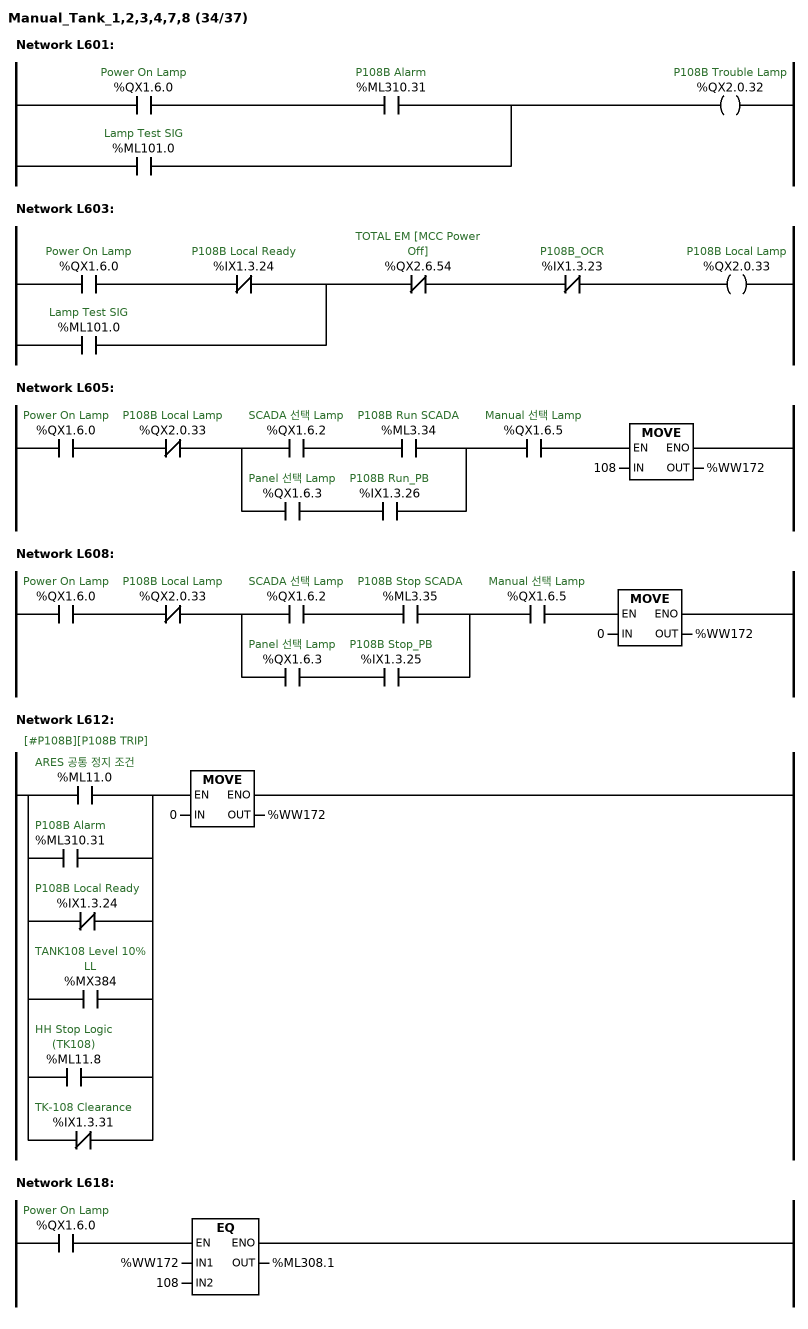
(* [picture p48: Manual_Tank_1,2,3,4,7,8 rungs L601-L618] *)
(* Rung L601 *)
%QX2.0.32 := (%QX1.6.0 AND %ML310.31) OR %ML101.0;
(* Rung L603 *)
%QX2.0.33 := ((%QX1.6.0 AND NOT %IX1.3.24) OR %ML101.0) AND NOT %QX2.6.54 AND NOT %IX1.3.23;
(* Rung L605 *)
IF %QX1.6.0 AND NOT %QX2.0.33 AND ((%QX1.6.2 AND %ML3.34) OR (%QX1.6.3 AND %IX1.3.26)) AND %QX1.6.5 THEN
    %WW172 := 108;
END_IF;
(* Rung L608 *)
IF %QX1.6.0 AND NOT %QX2.0.33 AND ((%QX1.6.2 AND %ML3.35) OR (%QX1.6.3 AND %IX1.3.25)) AND %QX1.6.5 THEN
    %WW172 := 0;
END_IF;
(* [#P108B][P108B TRIP] *)
(* Rung L612 *)
IF %ML11.0 OR %ML310.31 OR NOT %IX1.3.24 OR %MX384 OR %ML11.8 OR NOT %IX1.3.31 THEN %WW172 := 0; END_IF;
(* Rung L618 *)
IF %QX1.6.0 THEN %ML308.1 := %WW172 = 108; END_IF;

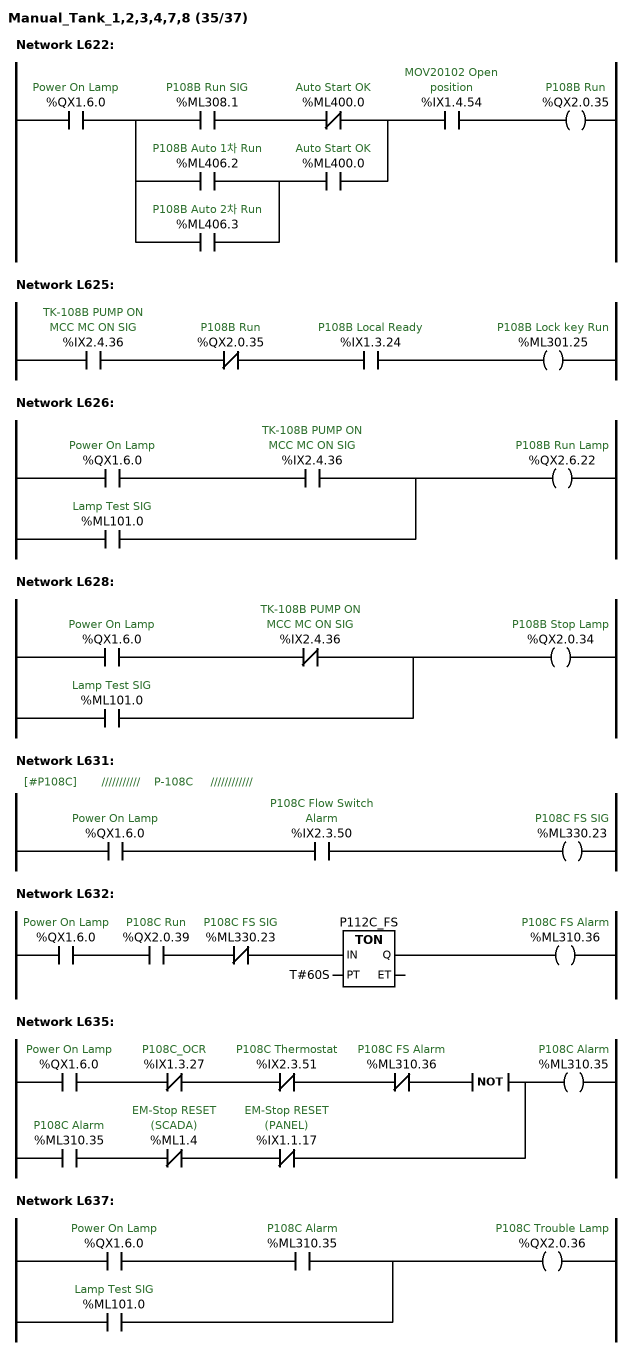
(* Rung L622 *)
%QX2.0.35 := %QX1.6.0 AND ((%ML308.1 AND NOT %ML400.0) OR ((%ML406.2 OR %ML406.3) AND %ML400.0)) AND %IX1.4.54;
(* Rung L625 *)
%ML301.25 := %IX2.4.36 AND NOT %QX2.0.35 AND %IX1.3.24;
(* Rung L626 *)
%QX2.6.22 := (%QX1.6.0 AND %IX2.4.36) OR %ML101.0;
(* Rung L628 *)
%QX2.0.34 := (%QX1.6.0 AND NOT %IX2.4.36) OR %ML101.0;
(* [#P108C]       ///////////    P-108C     //////////// *)
(* Rung L631 *)
%ML330.23 := %QX1.6.0 AND %IX2.3.50;
(* Rung L632 *)
P112C_FS(IN := %QX1.6.0 AND %QX2.0.39 AND NOT %ML330.23, PT := T#60S);
%ML310.36 := P112C_FS.Q;
(* Rung L635 *)
%ML310.35 := NOT (%QX1.6.0 AND NOT %IX1.3.27 AND NOT %IX2.3.51 AND NOT %ML310.36) OR (%ML310.35 AND NOT %ML1.4 AND NOT %IX1.1.17);
(* Rung L637 *)
%QX2.0.36 := (%QX1.6.0 AND %ML310.35) OR %ML101.0;

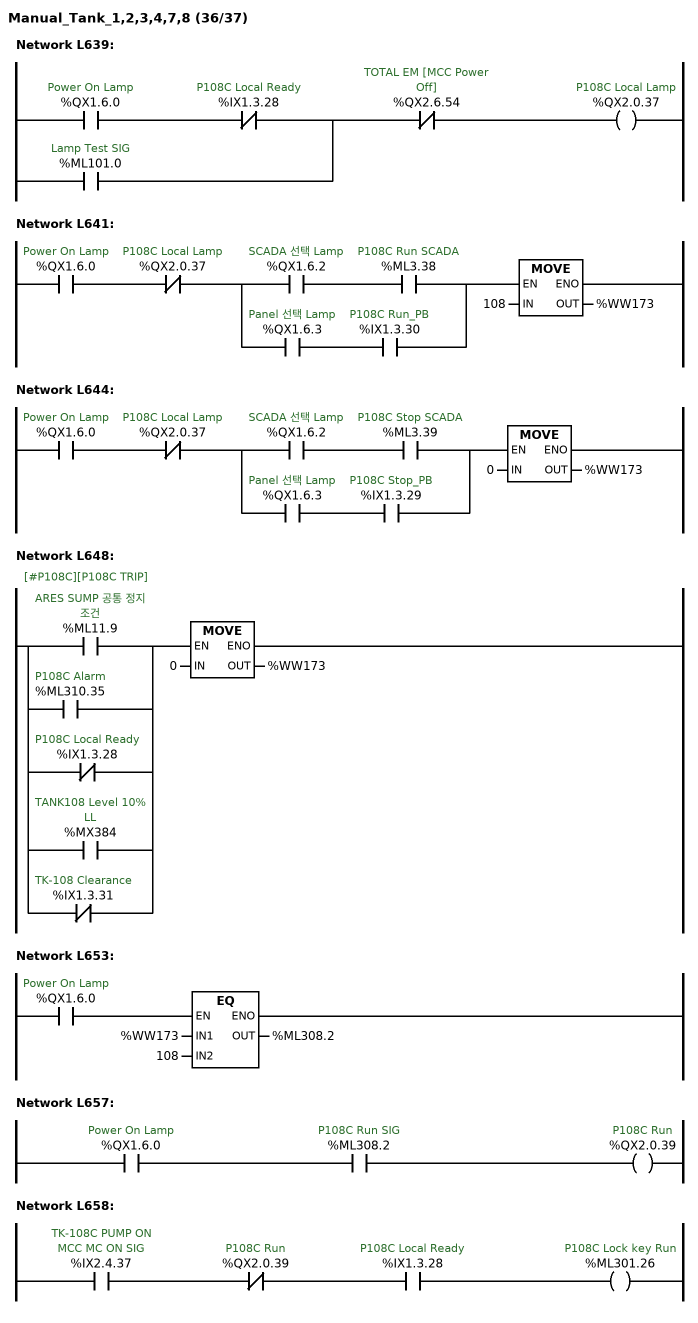
(* Rung L639 *)
%QX2.0.37 := ((%QX1.6.0 AND NOT %IX1.3.28) OR %ML101.0) AND NOT %QX2.6.54;
(* Rung L641 *)
IF %QX1.6.0 AND NOT %QX2.0.37 AND ((%QX1.6.2 AND %ML3.38) OR (%QX1.6.3 AND %IX1.3.30)) THEN
    %WW173 := 108;
END_IF;
(* Rung L644 *)
IF %QX1.6.0 AND NOT %QX2.0.37 AND ((%QX1.6.2 AND %ML3.39) OR (%QX1.6.3 AND %IX1.3.29)) THEN
    %WW173 := 0;
END_IF;
(* [#P108C][P108C TRIP] *)
(* Rung L648 *)
IF %ML11.9 OR %ML310.35 OR NOT %IX1.3.28 OR %MX384 OR NOT %IX1.3.31 THEN %WW173 := 0; END_IF;
(* Rung L653 *)
IF %QX1.6.0 THEN %ML308.2 := %WW173 = 108; END_IF;
(* Rung L657 *)
%QX2.0.39 := %QX1.6.0 AND %ML308.2;
(* Rung L658 *)
%ML301.26 := %IX2.4.37 AND NOT %QX2.0.39 AND %IX1.3.28;

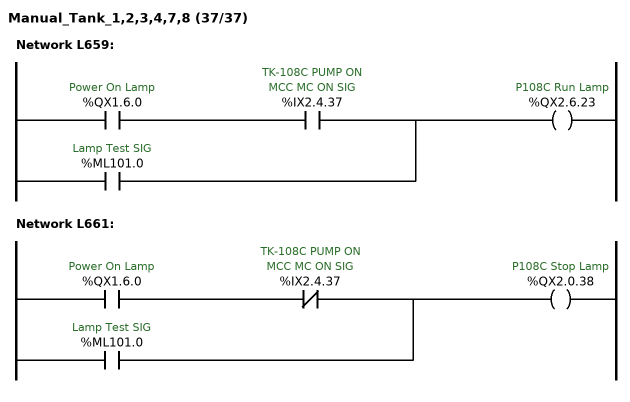
(* Rung L659 *)
%QX2.6.23 := (%QX1.6.0 AND %IX2.4.37) OR %ML101.0;
(* Rung L661 *)
%QX2.0.38 := (%QX1.6.0 AND NOT %IX2.4.37) OR %ML101.0;
END_PROGRAM

PROGRAM Manual_Tank_5,6,9,10 (* task: 스캔 프로그램 *)
VAR
    P105A_FS : TON;
    P105B_FS : TON;
    P105C_FS : TON;
    P106A_FS : TON;
    P106B_FS : TON;
    P106C_FS : TON;
    P109A_FS : TON;
    P109B_FS : TON;
    P109C_FS : TON;
    P110A_FS : TON;
    P110B_FS : TON;
    P110C_FS : TON;
END_VAR

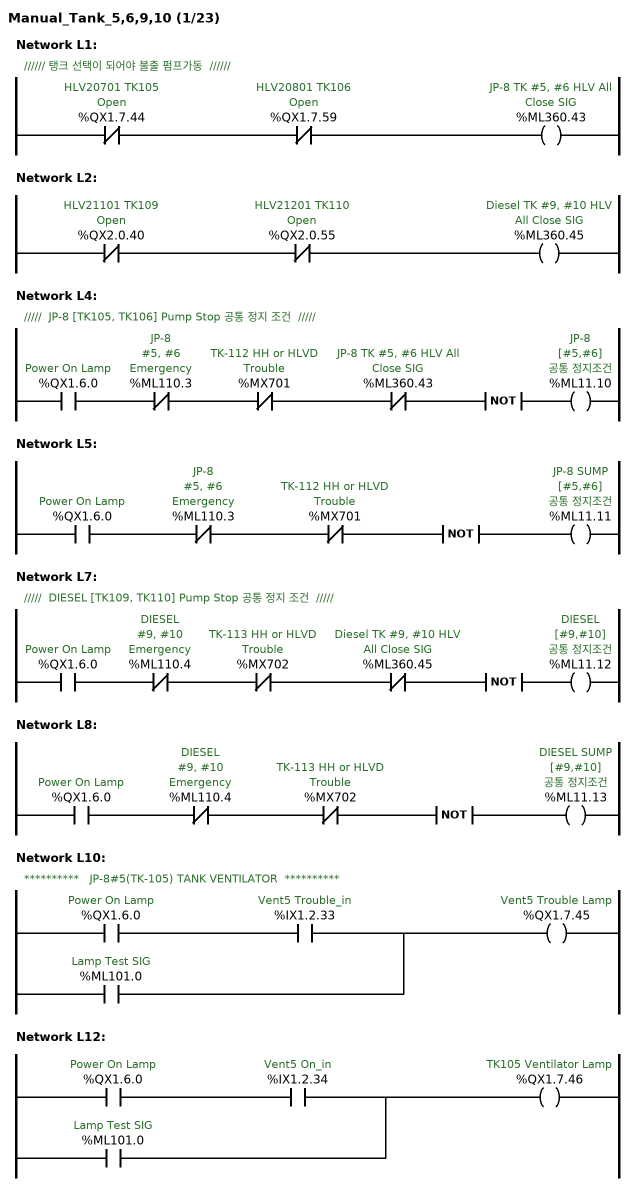
(* ////// 탱크 선택이 되어야 불출 펌프가동  ////// *)
(* Rung L1 *)
%ML360.43 := NOT %QX1.7.44 AND NOT %QX1.7.59;
(* Rung L2 *)
%ML360.45 := NOT %QX2.0.40 AND NOT %QX2.0.55;
(* /////  JP-8 [TK105, TK106] Pump Stop 공통 정지 조건  ///// *)
(* Rung L4 *)
%ML11.10 := NOT (%QX1.6.0 AND NOT %ML110.3 AND NOT %MX701 AND NOT %ML360.43);
(* Rung L5 *)
%ML11.11 := NOT (%QX1.6.0 AND NOT %ML110.3 AND NOT %MX701);
(* /////  DIESEL [TK109, TK110] Pump Stop 공통 정지 조건  ///// *)
(* Rung L7 *)
%ML11.12 := NOT (%QX1.6.0 AND NOT %ML110.4 AND NOT %MX702 AND NOT %ML360.45);
(* Rung L8 *)
%ML11.13 := NOT (%QX1.6.0 AND NOT %ML110.4 AND NOT %MX702);
(* **********   JP-8#5(TK-105) TANK VENTILATOR  ********** *)
(* Rung L10 *)
%QX1.7.45 := (%QX1.6.0 AND %IX1.2.33) OR %ML101.0;
(* Rung L12 *)
%QX1.7.46 := (%QX1.6.0 AND %IX1.2.34) OR %ML101.0;

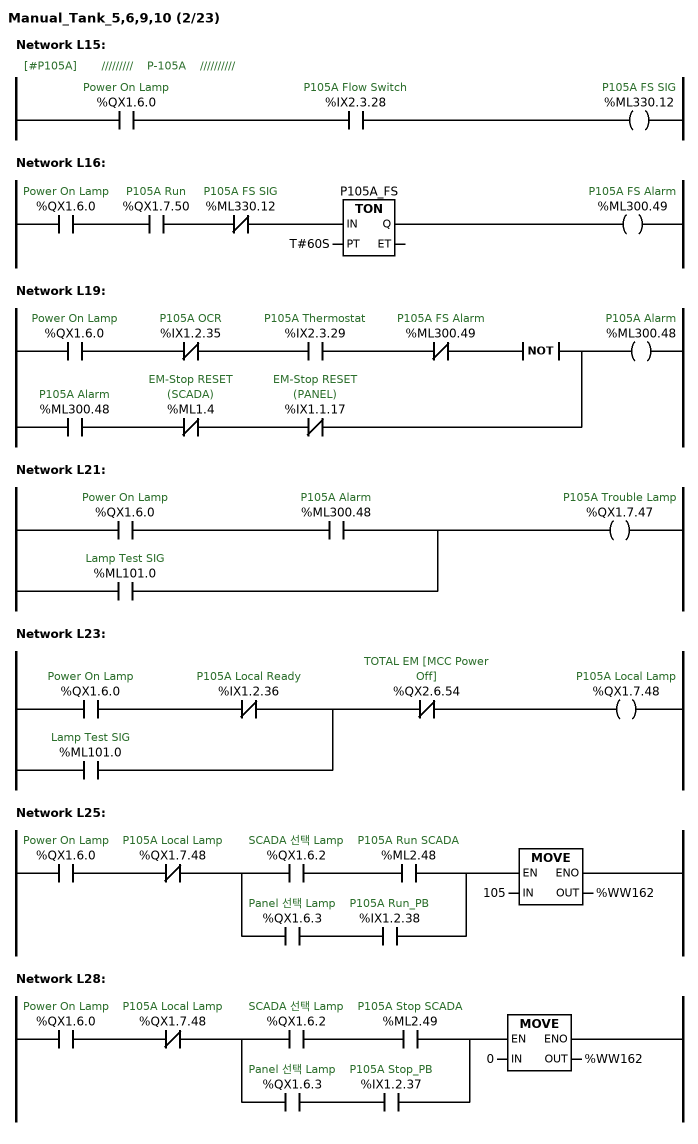
(* [#P105A]       /////////    P-105A    ////////// *)
(* Rung L15 *)
%ML330.12 := %QX1.6.0 AND %IX2.3.28;
(* Rung L16 *)
P105A_FS(IN := %QX1.6.0 AND %QX1.7.50 AND NOT %ML330.12, PT := T#60S);
%ML300.49 := P105A_FS.Q;
(* Rung L19 *)
%ML300.48 := NOT (%QX1.6.0 AND NOT %IX1.2.35 AND %IX2.3.29 AND NOT %ML300.49) OR (%ML300.48 AND NOT %ML1.4 AND NOT %IX1.1.17);
(* Rung L21 *)
%QX1.7.47 := (%QX1.6.0 AND %ML300.48) OR %ML101.0;
(* Rung L23 *)
%QX1.7.48 := ((%QX1.6.0 AND NOT %IX1.2.36) OR %ML101.0) AND NOT %QX2.6.54;
(* Rung L25 *)
IF %QX1.6.0 AND NOT %QX1.7.48 AND ((%QX1.6.2 AND %ML2.48) OR (%QX1.6.3 AND %IX1.2.38)) THEN
    %WW162 := 105;
END_IF;
(* Rung L28 *)
IF %QX1.6.0 AND NOT %QX1.7.48 AND ((%QX1.6.2 AND %ML2.49) OR (%QX1.6.3 AND %IX1.2.37)) THEN
    %WW162 := 0;
END_IF;

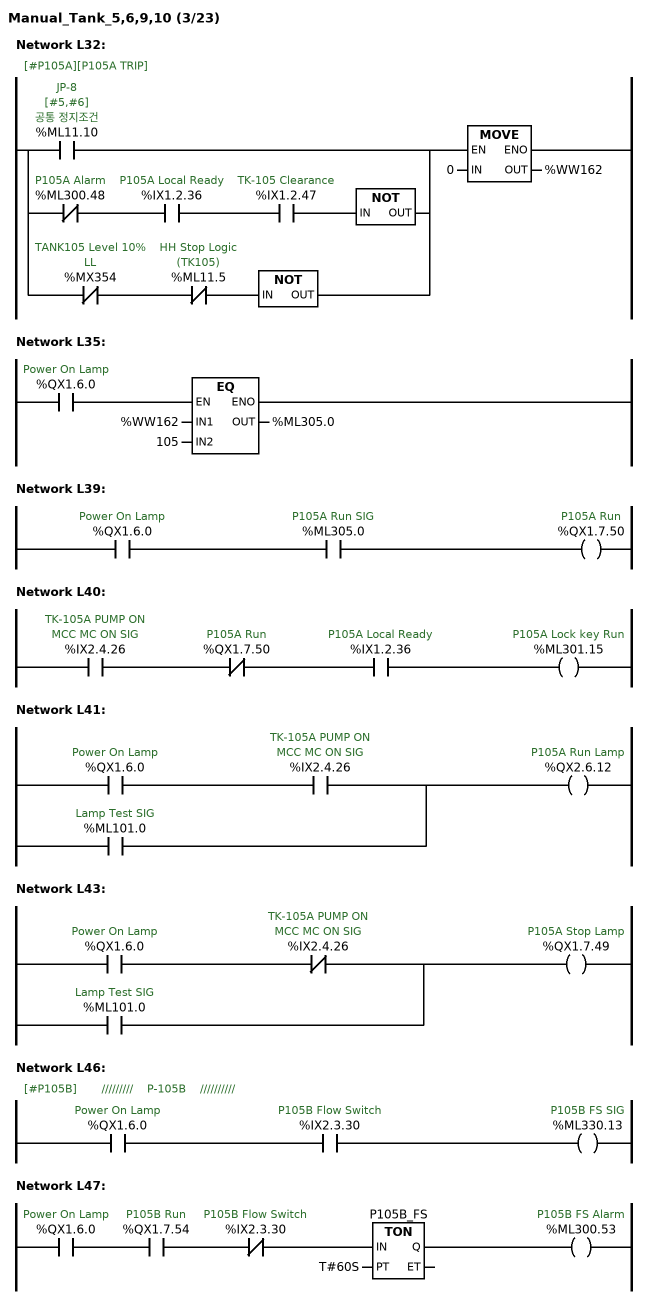
(* [#P105A][P105A TRIP] *)
(* Rung L32 *)
IF %ML11.10 OR (NOT (NOT %ML300.48 AND %IX1.2.36 AND %IX1.2.47)) OR (NOT (NOT %MX354 AND NOT %ML11.5)) THEN
    %WW162 := 0;
END_IF;
(* Rung L35 *)
IF %QX1.6.0 THEN %ML305.0 := %WW162 = 105; END_IF;
(* Rung L39 *)
%QX1.7.50 := %QX1.6.0 AND %ML305.0;
(* Rung L40 *)
%ML301.15 := %IX2.4.26 AND NOT %QX1.7.50 AND %IX1.2.36;
(* Rung L41 *)
%QX2.6.12 := (%QX1.6.0 AND %IX2.4.26) OR %ML101.0;
(* Rung L43 *)
%QX1.7.49 := (%QX1.6.0 AND NOT %IX2.4.26) OR %ML101.0;
(* [#P105B]       /////////    P-105B    ////////// *)
(* Rung L46 *)
%ML330.13 := %QX1.6.0 AND %IX2.3.30;
(* Rung L47 *)
P105B_FS(IN := %QX1.6.0 AND %QX1.7.54 AND NOT %IX2.3.30, PT := T#60S);
%ML300.53 := P105B_FS.Q;

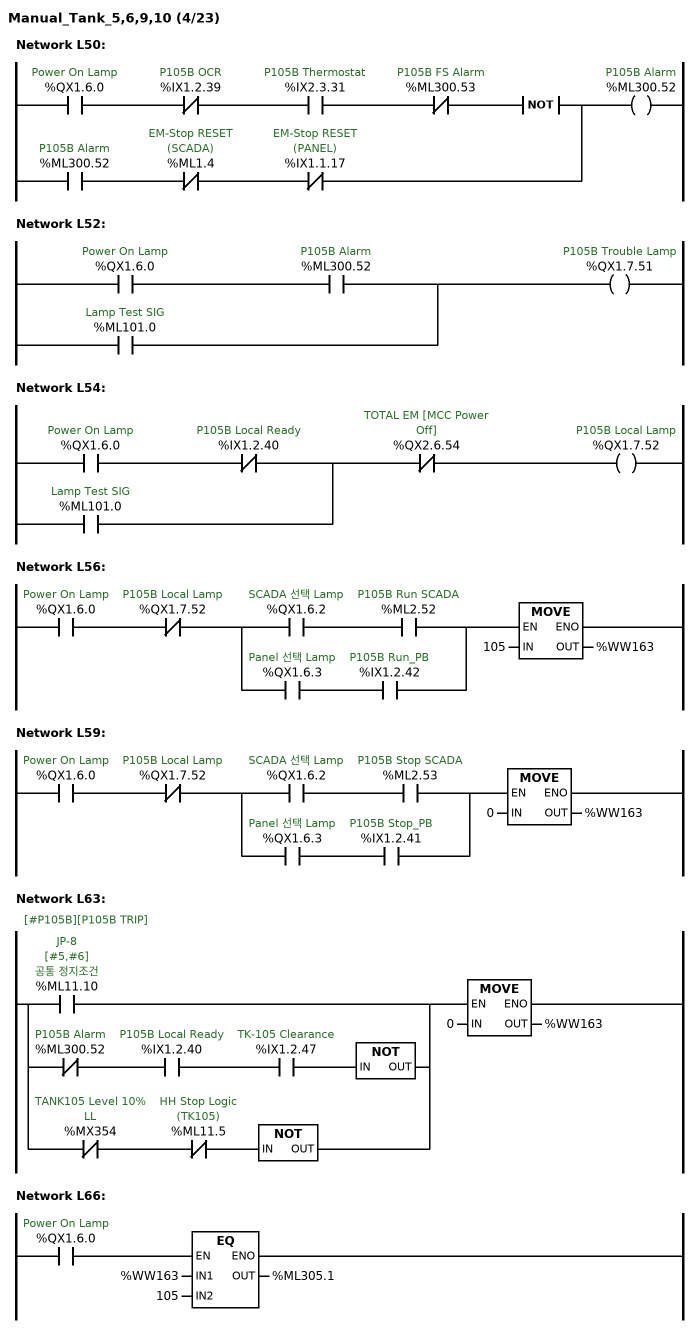
(* Rung L50 *)
%ML300.52 := NOT (%QX1.6.0 AND NOT %IX1.2.39 AND %IX2.3.31 AND NOT %ML300.53) OR (%ML300.52 AND NOT %ML1.4 AND NOT %IX1.1.17);
(* Rung L52 *)
%QX1.7.51 := (%QX1.6.0 AND %ML300.52) OR %ML101.0;
(* Rung L54 *)
%QX1.7.52 := ((%QX1.6.0 AND NOT %IX1.2.40) OR %ML101.0) AND NOT %QX2.6.54;
(* Rung L56 *)
IF %QX1.6.0 AND NOT %QX1.7.52 AND ((%QX1.6.2 AND %ML2.52) OR (%QX1.6.3 AND %IX1.2.42)) THEN
    %WW163 := 105;
END_IF;
(* Rung L59 *)
IF %QX1.6.0 AND NOT %QX1.7.52 AND ((%QX1.6.2 AND %ML2.53) OR (%QX1.6.3 AND %IX1.2.41)) THEN
    %WW163 := 0;
END_IF;
(* [#P105B][P105B TRIP] *)
(* Rung L63 *)
IF %ML11.10 OR (NOT (NOT %ML300.52 AND %IX1.2.40 AND %IX1.2.47)) OR (NOT (NOT %MX354 AND NOT %ML11.5)) THEN
    %WW163 := 0;
END_IF;
(* Rung L66 *)
IF %QX1.6.0 THEN %ML305.1 := %WW163 = 105; END_IF;

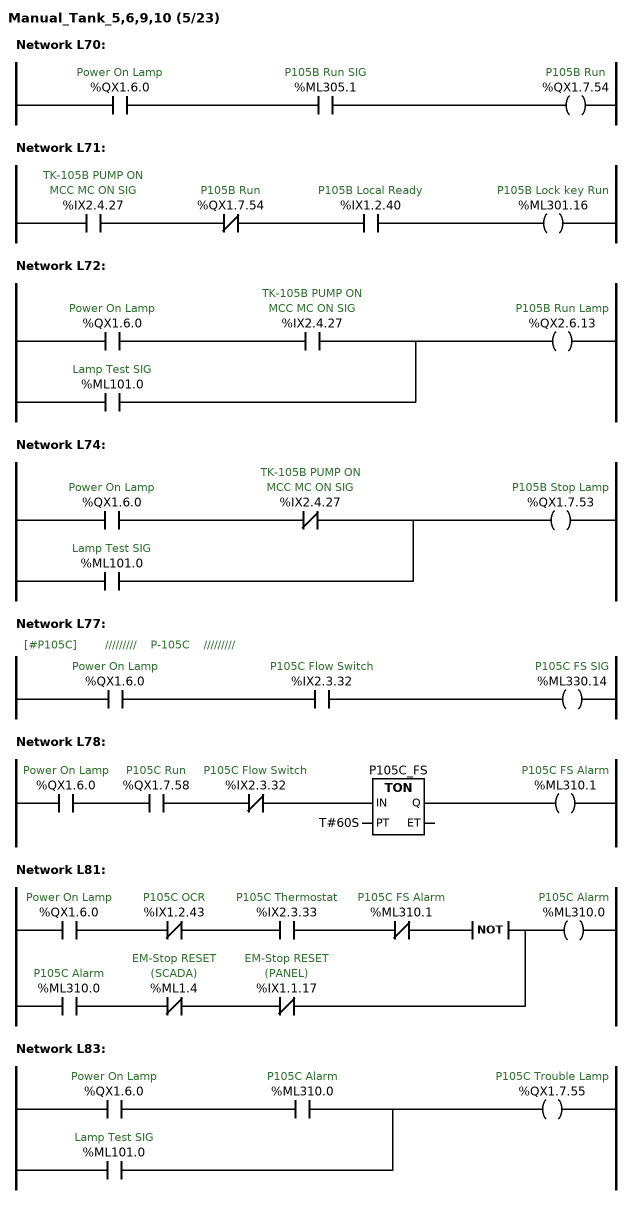
(* Rung L70 *)
%QX1.7.54 := %QX1.6.0 AND %ML305.1;
(* Rung L71 *)
%ML301.16 := %IX2.4.27 AND NOT %QX1.7.54 AND %IX1.2.40;
(* Rung L72 *)
%QX2.6.13 := (%QX1.6.0 AND %IX2.4.27) OR %ML101.0;
(* Rung L74 *)
%QX1.7.53 := (%QX1.6.0 AND NOT %IX2.4.27) OR %ML101.0;
(* [#P105C]        /////////    P-105C    ///////// *)
(* Rung L77 *)
%ML330.14 := %QX1.6.0 AND %IX2.3.32;
(* Rung L78 *)
P105C_FS(IN := %QX1.6.0 AND %QX1.7.58 AND NOT %IX2.3.32, PT := T#60S);
%ML310.1 := P105C_FS.Q;
(* Rung L81 *)
%ML310.0 := NOT (%QX1.6.0 AND NOT %IX1.2.43 AND %IX2.3.33 AND NOT %ML310.1) OR (%ML310.0 AND NOT %ML1.4 AND NOT %IX1.1.17);
(* Rung L83 *)
%QX1.7.55 := (%QX1.6.0 AND %ML310.0) OR %ML101.0;

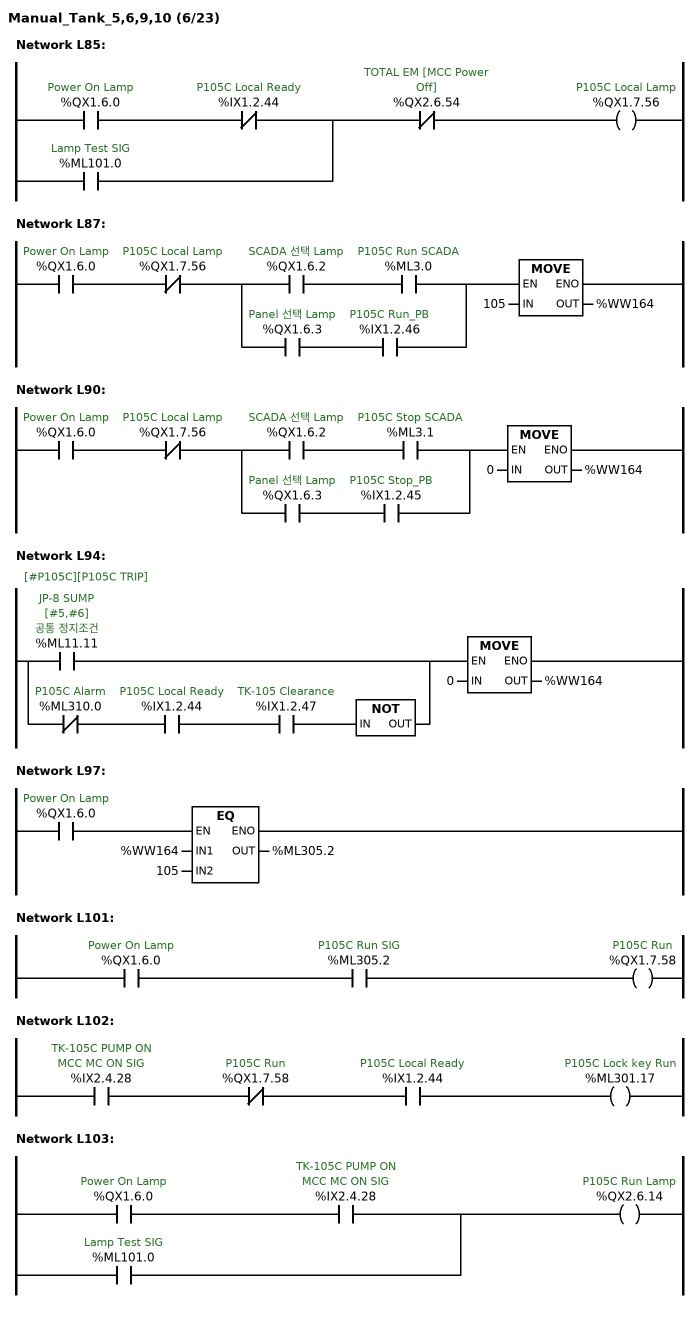
(* Rung L85 *)
%QX1.7.56 := ((%QX1.6.0 AND NOT %IX1.2.44) OR %ML101.0) AND NOT %QX2.6.54;
(* Rung L87 *)
IF %QX1.6.0 AND NOT %QX1.7.56 AND ((%QX1.6.2 AND %ML3.0) OR (%QX1.6.3 AND %IX1.2.46)) THEN
    %WW164 := 105;
END_IF;
(* Rung L90 *)
IF %QX1.6.0 AND NOT %QX1.7.56 AND ((%QX1.6.2 AND %ML3.1) OR (%QX1.6.3 AND %IX1.2.45)) THEN
    %WW164 := 0;
END_IF;
(* [#P105C][P105C TRIP] *)
(* Rung L94 *)
IF %ML11.11 OR (NOT (NOT %ML310.0 AND %IX1.2.44 AND %IX1.2.47)) THEN %WW164 := 0; END_IF;
(* Rung L97 *)
IF %QX1.6.0 THEN %ML305.2 := %WW164 = 105; END_IF;
(* Rung L101 *)
%QX1.7.58 := %QX1.6.0 AND %ML305.2;
(* Rung L102 *)
%ML301.17 := %IX2.4.28 AND NOT %QX1.7.58 AND %IX1.2.44;
(* Rung L103 *)
%QX2.6.14 := (%QX1.6.0 AND %IX2.4.28) OR %ML101.0;

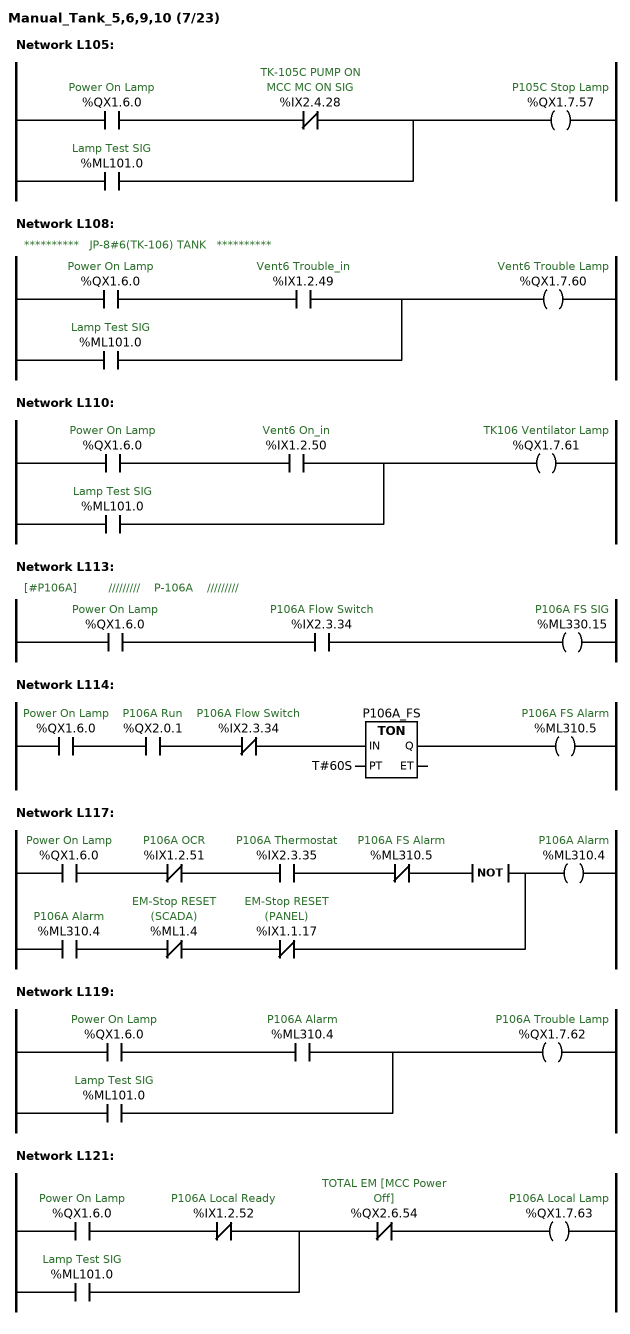
(* Rung L105 *)
%QX1.7.57 := (%QX1.6.0 AND NOT %IX2.4.28) OR %ML101.0;
(* **********   JP-8#6(TK-106) TANK   ********** *)
(* Rung L108 *)
%QX1.7.60 := (%QX1.6.0 AND %IX1.2.49) OR %ML101.0;
(* Rung L110 *)
%QX1.7.61 := (%QX1.6.0 AND %IX1.2.50) OR %ML101.0;
(* [#P106A]         /////////    P-106A    ///////// *)
(* Rung L113 *)
%ML330.15 := %QX1.6.0 AND %IX2.3.34;
(* Rung L114 *)
P106A_FS(IN := %QX1.6.0 AND %QX2.0.1 AND NOT %IX2.3.34, PT := T#60S);
%ML310.5 := P106A_FS.Q;
(* Rung L117 *)
%ML310.4 := NOT (%QX1.6.0 AND NOT %IX1.2.51 AND %IX2.3.35 AND NOT %ML310.5) OR (%ML310.4 AND NOT %ML1.4 AND NOT %IX1.1.17);
(* Rung L119 *)
%QX1.7.62 := (%QX1.6.0 AND %ML310.4) OR %ML101.0;
(* Rung L121 *)
%QX1.7.63 := ((%QX1.6.0 AND NOT %IX1.2.52) OR %ML101.0) AND NOT %QX2.6.54;

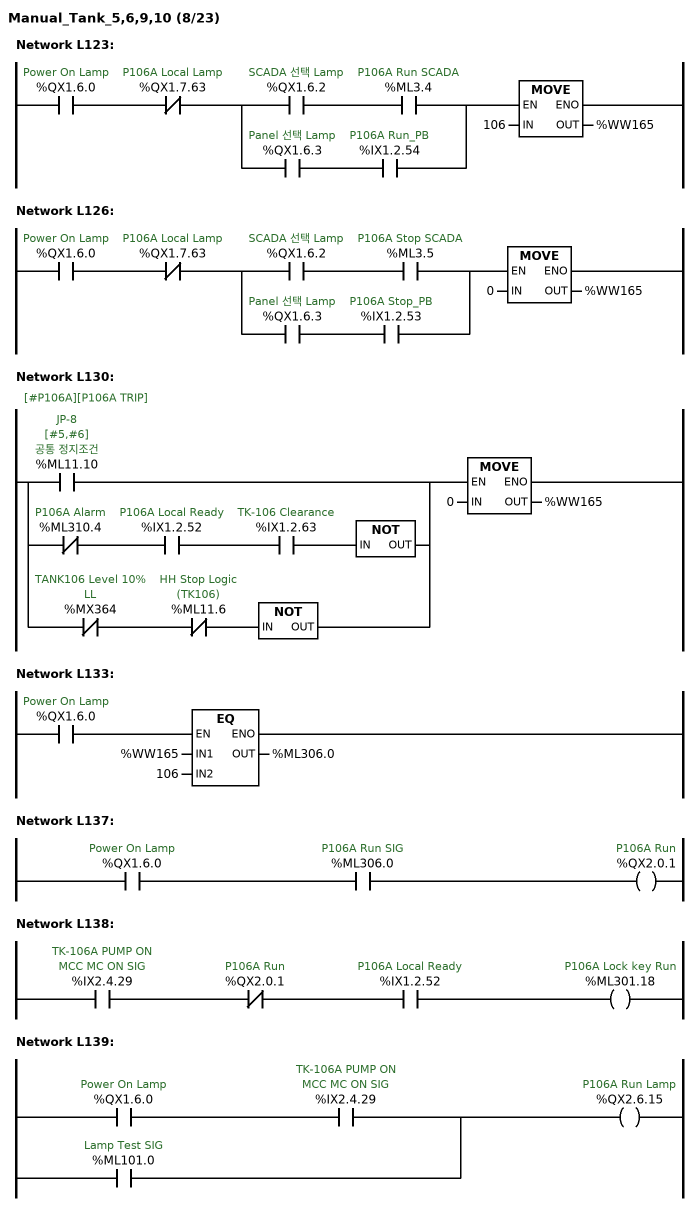
(* Rung L123 *)
IF %QX1.6.0 AND NOT %QX1.7.63 AND ((%QX1.6.2 AND %ML3.4) OR (%QX1.6.3 AND %IX1.2.54)) THEN
    %WW165 := 106;
END_IF;
(* Rung L126 *)
IF %QX1.6.0 AND NOT %QX1.7.63 AND ((%QX1.6.2 AND %ML3.5) OR (%QX1.6.3 AND %IX1.2.53)) THEN
    %WW165 := 0;
END_IF;
(* [#P106A][P106A TRIP] *)
(* Rung L130 *)
IF %ML11.10 OR (NOT (NOT %ML310.4 AND %IX1.2.52 AND %IX1.2.63)) OR (NOT (NOT %MX364 AND NOT %ML11.6)) THEN
    %WW165 := 0;
END_IF;
(* Rung L133 *)
IF %QX1.6.0 THEN %ML306.0 := %WW165 = 106; END_IF;
(* Rung L137 *)
%QX2.0.1 := %QX1.6.0 AND %ML306.0;
(* Rung L138 *)
%ML301.18 := %IX2.4.29 AND NOT %QX2.0.1 AND %IX1.2.52;
(* Rung L139 *)
%QX2.6.15 := (%QX1.6.0 AND %IX2.4.29) OR %ML101.0;

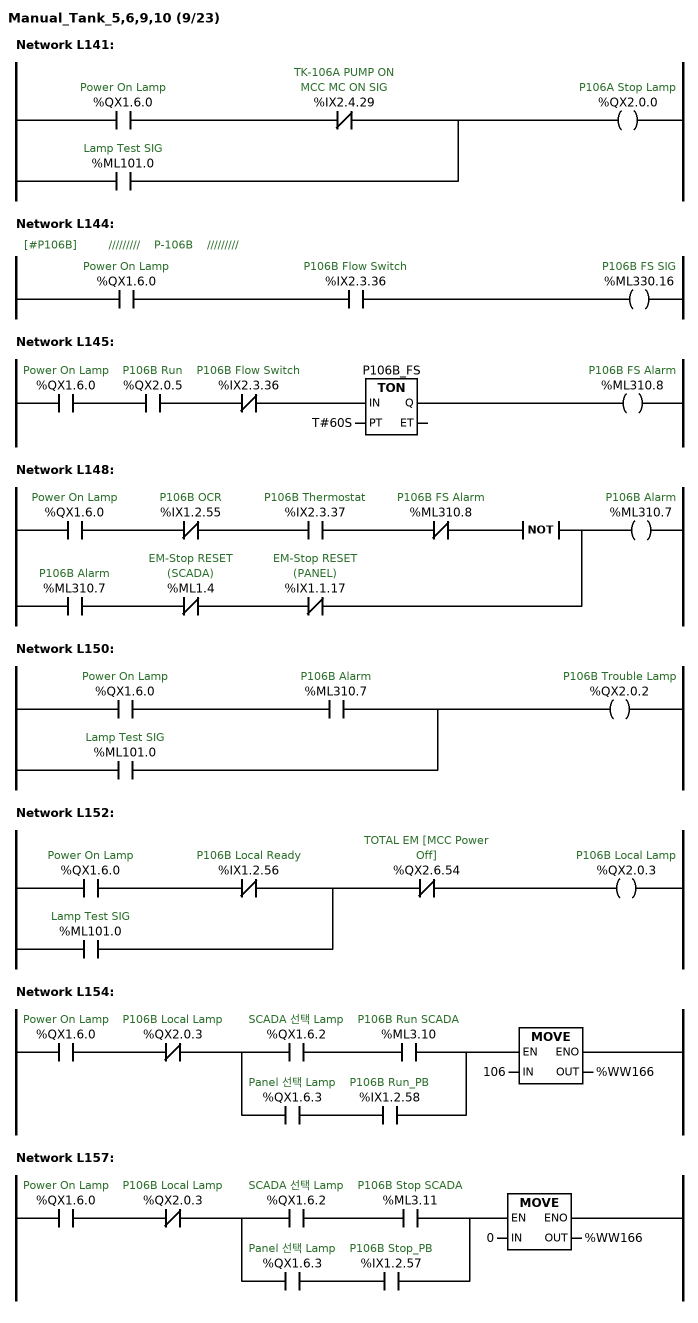
(* Rung L141 *)
%QX2.0.0 := (%QX1.6.0 AND NOT %IX2.4.29) OR %ML101.0;
(* [#P106B]         /////////    P-106B    ///////// *)
(* Rung L144 *)
%ML330.16 := %QX1.6.0 AND %IX2.3.36;
(* Rung L145 *)
P106B_FS(IN := %QX1.6.0 AND %QX2.0.5 AND NOT %IX2.3.36, PT := T#60S);
%ML310.8 := P106B_FS.Q;
(* Rung L148 *)
%ML310.7 := NOT (%QX1.6.0 AND NOT %IX1.2.55 AND %IX2.3.37 AND NOT %ML310.8) OR (%ML310.7 AND NOT %ML1.4 AND NOT %IX1.1.17);
(* Rung L150 *)
%QX2.0.2 := (%QX1.6.0 AND %ML310.7) OR %ML101.0;
(* Rung L152 *)
%QX2.0.3 := ((%QX1.6.0 AND NOT %IX1.2.56) OR %ML101.0) AND NOT %QX2.6.54;
(* Rung L154 *)
IF %QX1.6.0 AND NOT %QX2.0.3 AND ((%QX1.6.2 AND %ML3.10) OR (%QX1.6.3 AND %IX1.2.58)) THEN
    %WW166 := 106;
END_IF;
(* Rung L157 *)
IF %QX1.6.0 AND NOT %QX2.0.3 AND ((%QX1.6.2 AND %ML3.11) OR (%QX1.6.3 AND %IX1.2.57)) THEN
    %WW166 := 0;
END_IF;

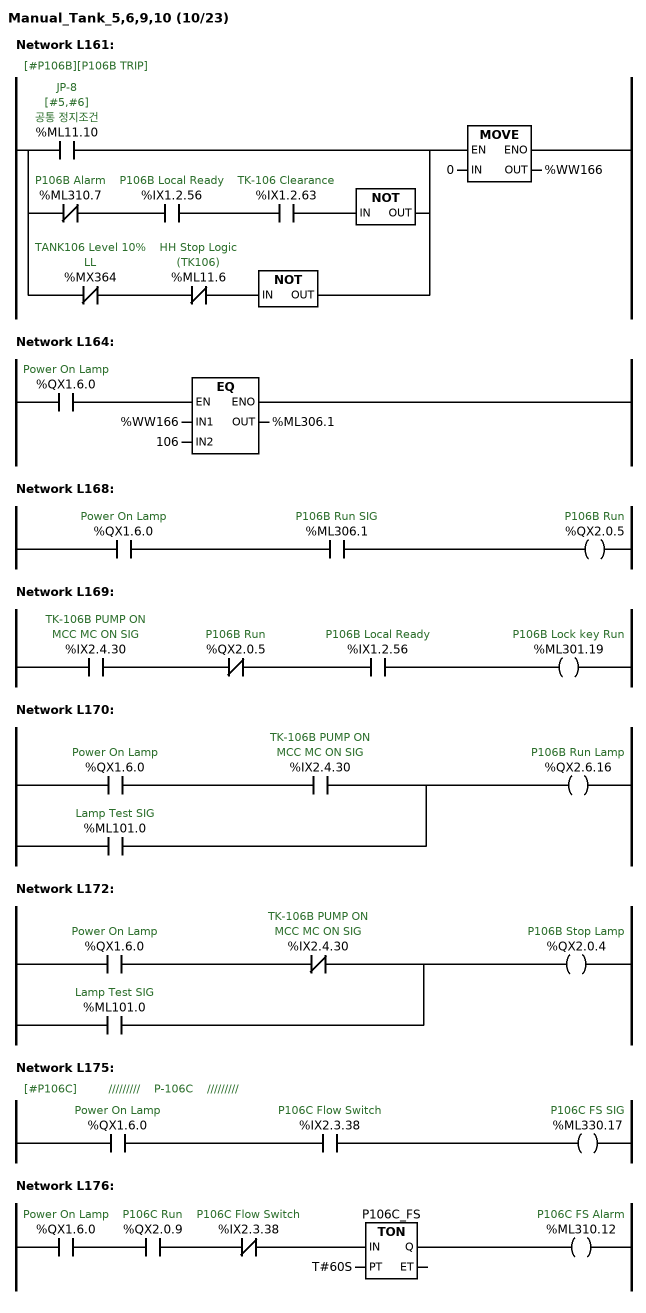
(* [#P106B][P106B TRIP] *)
(* Rung L161 *)
IF %ML11.10 OR (NOT (NOT %ML310.7 AND %IX1.2.56 AND %IX1.2.63)) OR (NOT (NOT %MX364 AND NOT %ML11.6)) THEN
    %WW166 := 0;
END_IF;
(* Rung L164 *)
IF %QX1.6.0 THEN %ML306.1 := %WW166 = 106; END_IF;
(* Rung L168 *)
%QX2.0.5 := %QX1.6.0 AND %ML306.1;
(* Rung L169 *)
%ML301.19 := %IX2.4.30 AND NOT %QX2.0.5 AND %IX1.2.56;
(* Rung L170 *)
%QX2.6.16 := (%QX1.6.0 AND %IX2.4.30) OR %ML101.0;
(* Rung L172 *)
%QX2.0.4 := (%QX1.6.0 AND NOT %IX2.4.30) OR %ML101.0;
(* [#P106C]         /////////    P-106C    ///////// *)
(* Rung L175 *)
%ML330.17 := %QX1.6.0 AND %IX2.3.38;
(* Rung L176 *)
P106C_FS(IN := %QX1.6.0 AND %QX2.0.9 AND NOT %IX2.3.38, PT := T#60S);
%ML310.12 := P106C_FS.Q;

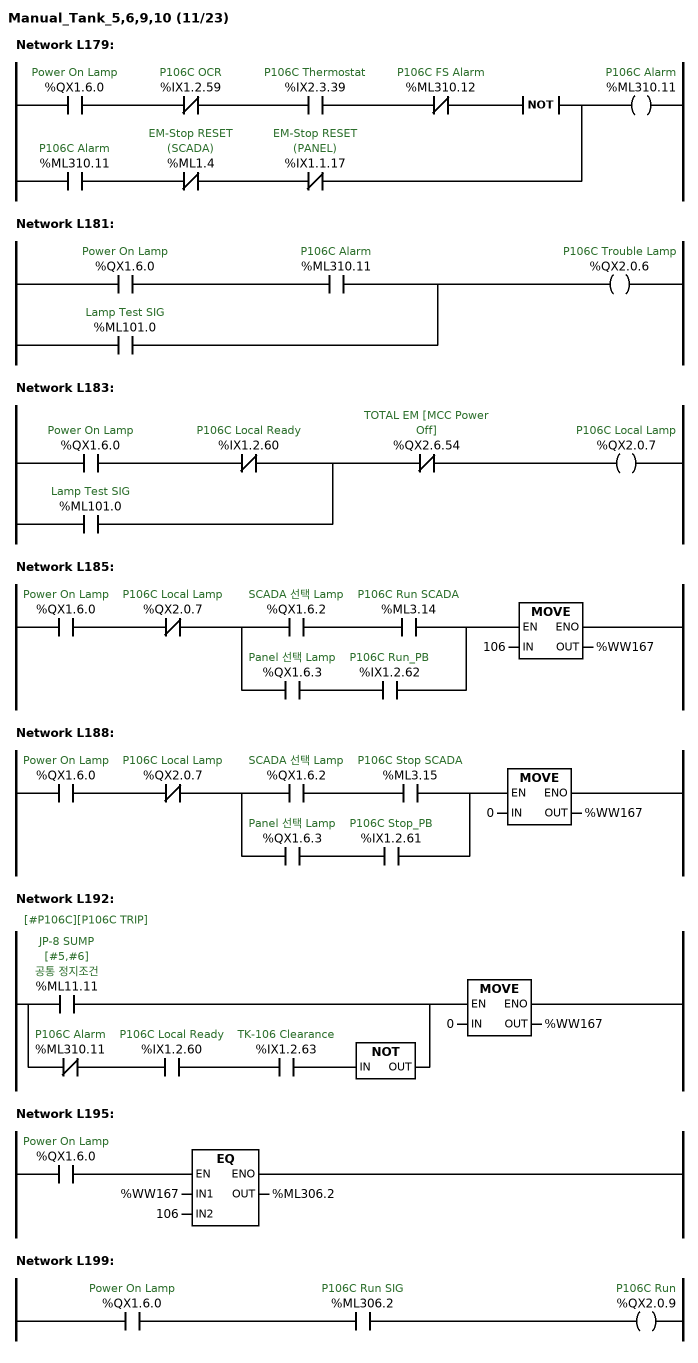
(* Rung L179 *)
%ML310.11 := NOT (%QX1.6.0 AND NOT %IX1.2.59 AND %IX2.3.39 AND NOT %ML310.12) OR (%ML310.11 AND NOT %ML1.4 AND NOT %IX1.1.17);
(* Rung L181 *)
%QX2.0.6 := (%QX1.6.0 AND %ML310.11) OR %ML101.0;
(* Rung L183 *)
%QX2.0.7 := ((%QX1.6.0 AND NOT %IX1.2.60) OR %ML101.0) AND NOT %QX2.6.54;
(* Rung L185 *)
IF %QX1.6.0 AND NOT %QX2.0.7 AND ((%QX1.6.2 AND %ML3.14) OR (%QX1.6.3 AND %IX1.2.62)) THEN
    %WW167 := 106;
END_IF;
(* Rung L188 *)
IF %QX1.6.0 AND NOT %QX2.0.7 AND ((%QX1.6.2 AND %ML3.15) OR (%QX1.6.3 AND %IX1.2.61)) THEN
    %WW167 := 0;
END_IF;
(* [#P106C][P106C TRIP] *)
(* Rung L192 *)
IF %ML11.11 OR (NOT (NOT %ML310.11 AND %IX1.2.60 AND %IX1.2.63)) THEN %WW167 := 0; END_IF;
(* Rung L195 *)
IF %QX1.6.0 THEN %ML306.2 := %WW167 = 106; END_IF;
(* Rung L199 *)
%QX2.0.9 := %QX1.6.0 AND %ML306.2;

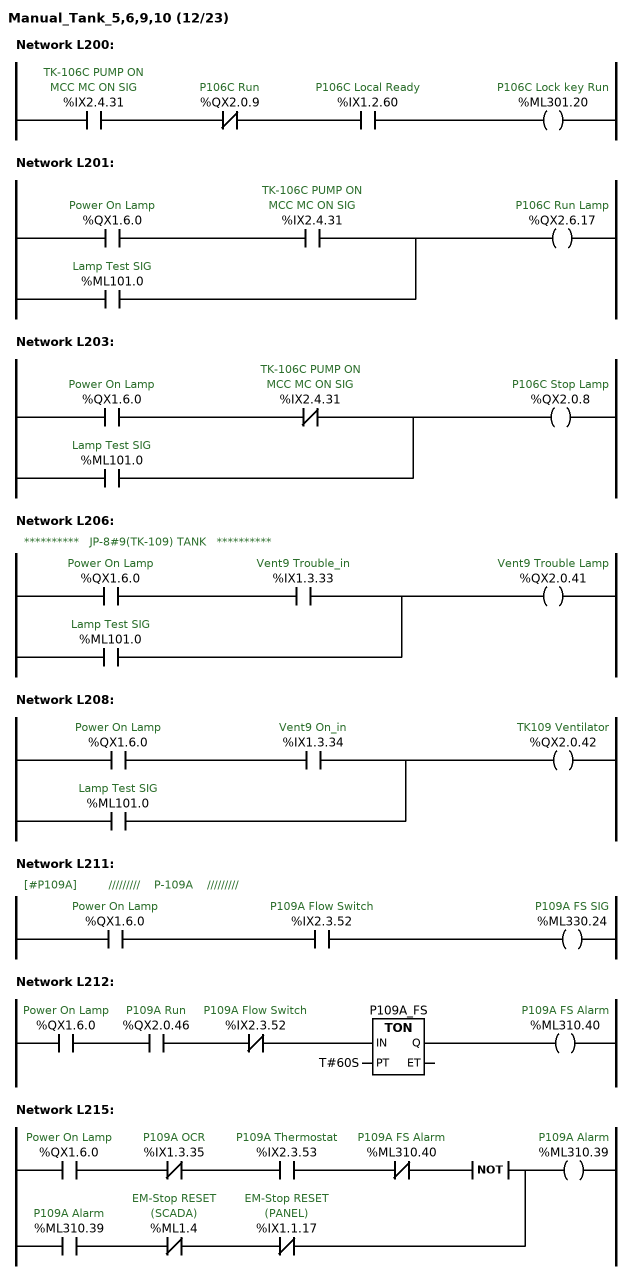
(* Rung L200 *)
%ML301.20 := %IX2.4.31 AND NOT %QX2.0.9 AND %IX1.2.60;
(* Rung L201 *)
%QX2.6.17 := (%QX1.6.0 AND %IX2.4.31) OR %ML101.0;
(* Rung L203 *)
%QX2.0.8 := (%QX1.6.0 AND NOT %IX2.4.31) OR %ML101.0;
(* **********   JP-8#9(TK-109) TANK   ********** *)
(* Rung L206 *)
%QX2.0.41 := (%QX1.6.0 AND %IX1.3.33) OR %ML101.0;
(* Rung L208 *)
%QX2.0.42 := (%QX1.6.0 AND %IX1.3.34) OR %ML101.0;
(* [#P109A]         /////////    P-109A    ///////// *)
(* Rung L211 *)
%ML330.24 := %QX1.6.0 AND %IX2.3.52;
(* Rung L212 *)
P109A_FS(IN := %QX1.6.0 AND %QX2.0.46 AND NOT %IX2.3.52, PT := T#60S);
%ML310.40 := P109A_FS.Q;
(* Rung L215 *)
%ML310.39 := NOT (%QX1.6.0 AND NOT %IX1.3.35 AND %IX2.3.53 AND NOT %ML310.40) OR (%ML310.39 AND NOT %ML1.4 AND NOT %IX1.1.17);

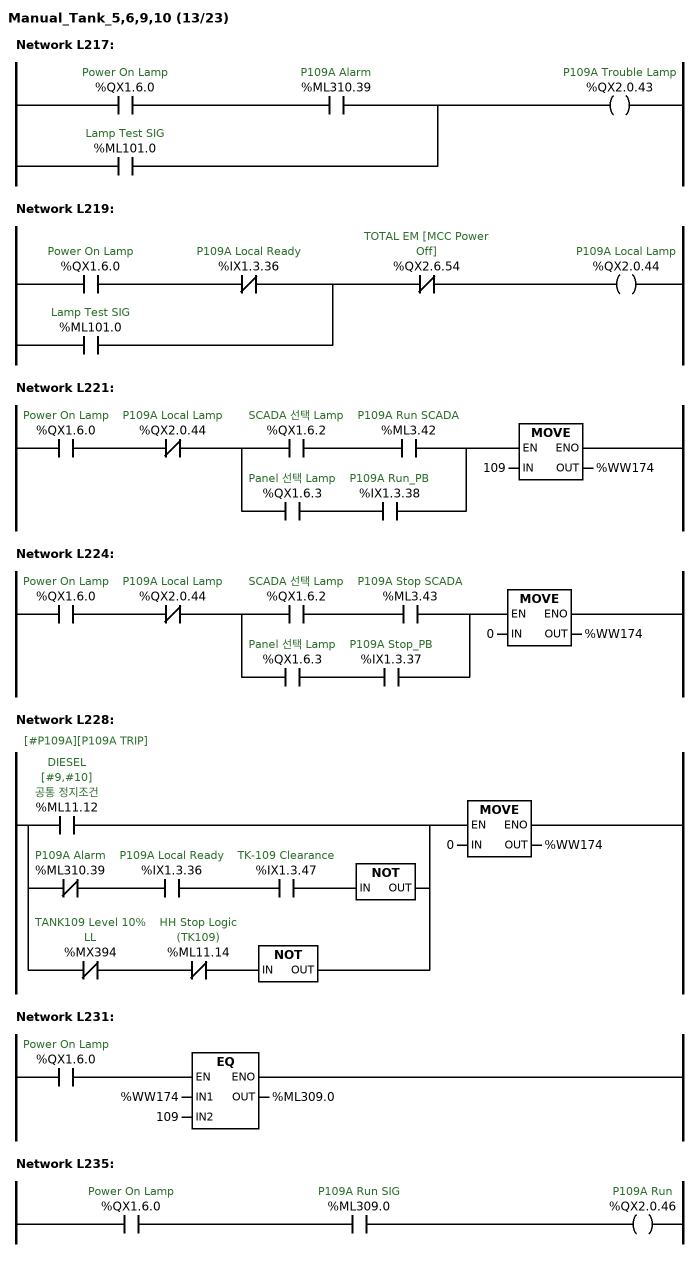
(* Rung L217 *)
%QX2.0.43 := (%QX1.6.0 AND %ML310.39) OR %ML101.0;
(* Rung L219 *)
%QX2.0.44 := ((%QX1.6.0 AND NOT %IX1.3.36) OR %ML101.0) AND NOT %QX2.6.54;
(* Rung L221 *)
IF %QX1.6.0 AND NOT %QX2.0.44 AND ((%QX1.6.2 AND %ML3.42) OR (%QX1.6.3 AND %IX1.3.38)) THEN
    %WW174 := 109;
END_IF;
(* Rung L224 *)
IF %QX1.6.0 AND NOT %QX2.0.44 AND ((%QX1.6.2 AND %ML3.43) OR (%QX1.6.3 AND %IX1.3.37)) THEN
    %WW174 := 0;
END_IF;
(* [#P109A][P109A TRIP] *)
(* Rung L228 *)
IF %ML11.12 OR (NOT (NOT %ML310.39 AND %IX1.3.36 AND %IX1.3.47)) OR (NOT (NOT %MX394 AND NOT %ML11.14)) THEN
    %WW174 := 0;
END_IF;
(* Rung L231 *)
IF %QX1.6.0 THEN %ML309.0 := %WW174 = 109; END_IF;
(* Rung L235 *)
%QX2.0.46 := %QX1.6.0 AND %ML309.0;

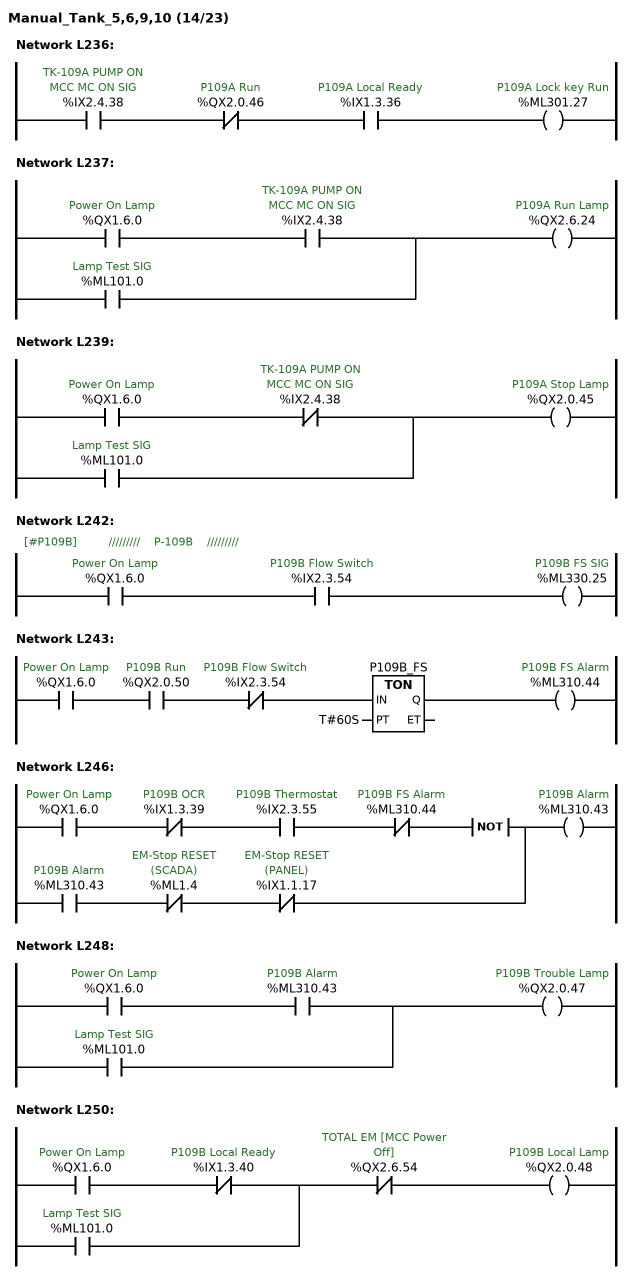
(* Rung L236 *)
%ML301.27 := %IX2.4.38 AND NOT %QX2.0.46 AND %IX1.3.36;
(* Rung L237 *)
%QX2.6.24 := (%QX1.6.0 AND %IX2.4.38) OR %ML101.0;
(* Rung L239 *)
%QX2.0.45 := (%QX1.6.0 AND NOT %IX2.4.38) OR %ML101.0;
(* [#P109B]         /////////    P-109B    ///////// *)
(* Rung L242 *)
%ML330.25 := %QX1.6.0 AND %IX2.3.54;
(* Rung L243 *)
P109B_FS(IN := %QX1.6.0 AND %QX2.0.50 AND NOT %IX2.3.54, PT := T#60S);
%ML310.44 := P109B_FS.Q;
(* Rung L246 *)
%ML310.43 := NOT (%QX1.6.0 AND NOT %IX1.3.39 AND %IX2.3.55 AND NOT %ML310.44) OR (%ML310.43 AND NOT %ML1.4 AND NOT %IX1.1.17);
(* Rung L248 *)
%QX2.0.47 := (%QX1.6.0 AND %ML310.43) OR %ML101.0;
(* Rung L250 *)
%QX2.0.48 := ((%QX1.6.0 AND NOT %IX1.3.40) OR %ML101.0) AND NOT %QX2.6.54;

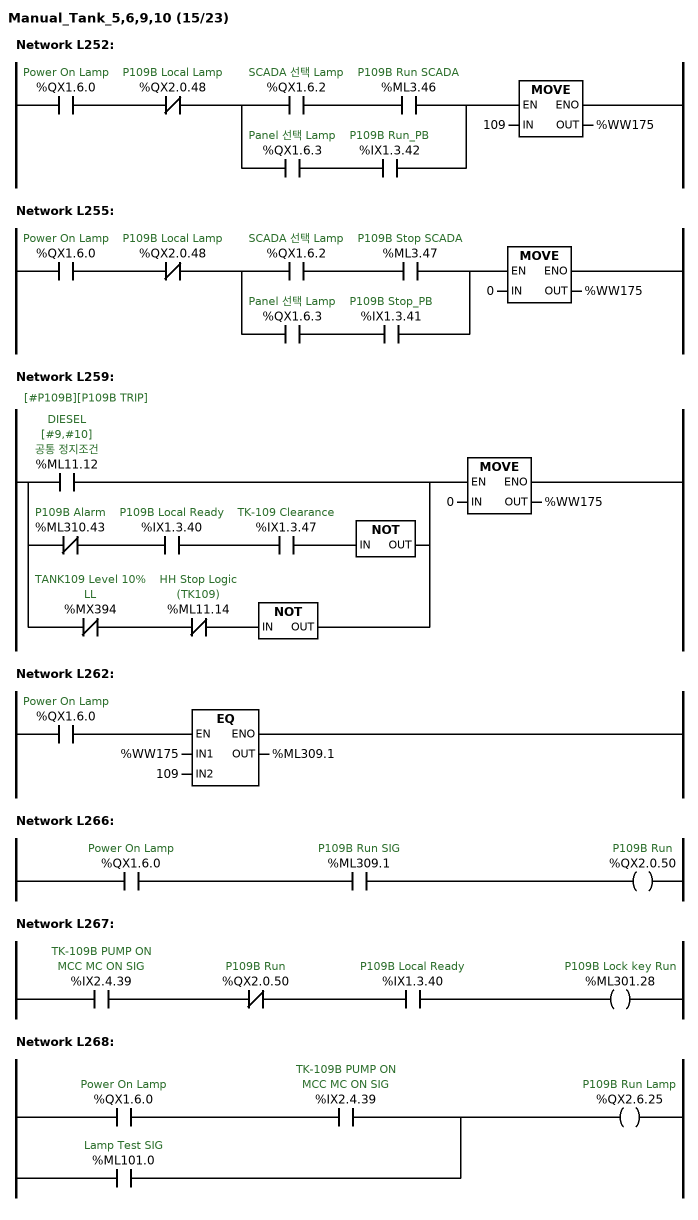
(* Rung L252 *)
IF %QX1.6.0 AND NOT %QX2.0.48 AND ((%QX1.6.2 AND %ML3.46) OR (%QX1.6.3 AND %IX1.3.42)) THEN
    %WW175 := 109;
END_IF;
(* Rung L255 *)
IF %QX1.6.0 AND NOT %QX2.0.48 AND ((%QX1.6.2 AND %ML3.47) OR (%QX1.6.3 AND %IX1.3.41)) THEN
    %WW175 := 0;
END_IF;
(* [#P109B][P109B TRIP] *)
(* Rung L259 *)
IF %ML11.12 OR (NOT (NOT %ML310.43 AND %IX1.3.40 AND %IX1.3.47)) OR (NOT (NOT %MX394 AND NOT %ML11.14)) THEN
    %WW175 := 0;
END_IF;
(* Rung L262 *)
IF %QX1.6.0 THEN %ML309.1 := %WW175 = 109; END_IF;
(* Rung L266 *)
%QX2.0.50 := %QX1.6.0 AND %ML309.1;
(* Rung L267 *)
%ML301.28 := %IX2.4.39 AND NOT %QX2.0.50 AND %IX1.3.40;
(* Rung L268 *)
%QX2.6.25 := (%QX1.6.0 AND %IX2.4.39) OR %ML101.0;

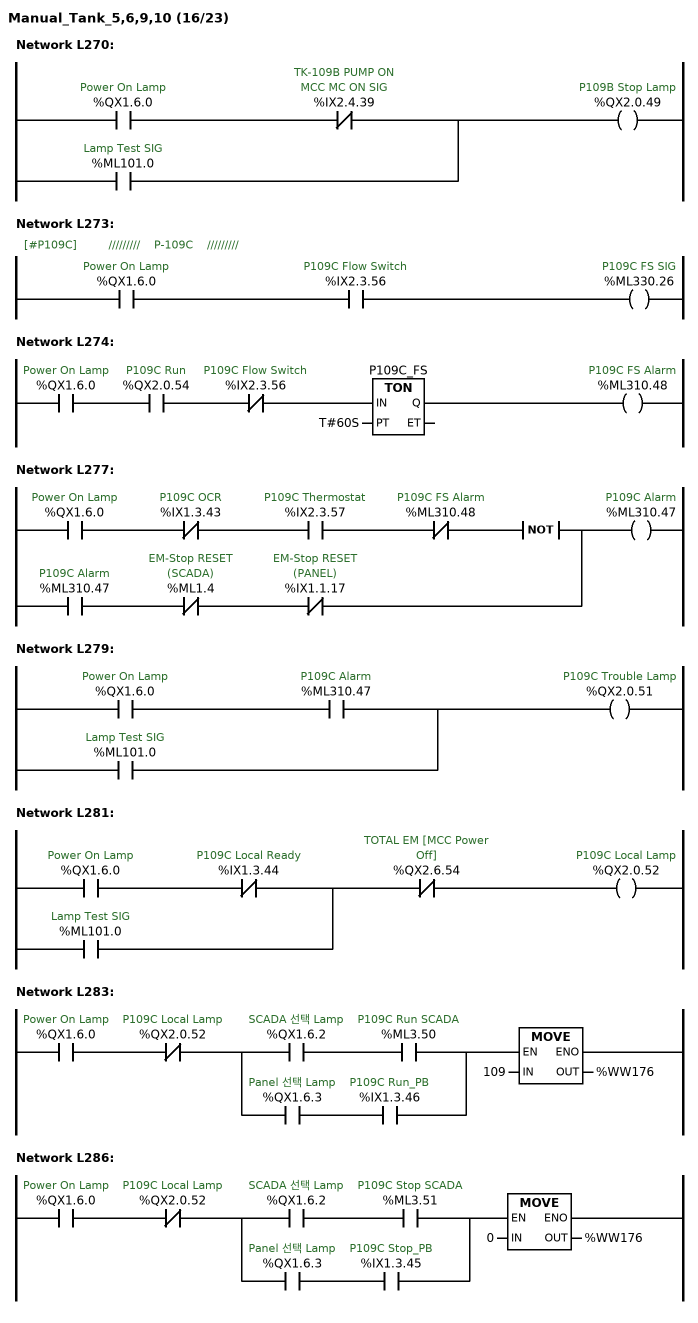
(* Rung L270 *)
%QX2.0.49 := (%QX1.6.0 AND NOT %IX2.4.39) OR %ML101.0;
(* [#P109C]         /////////    P-109C    ///////// *)
(* Rung L273 *)
%ML330.26 := %QX1.6.0 AND %IX2.3.56;
(* Rung L274 *)
P109C_FS(IN := %QX1.6.0 AND %QX2.0.54 AND NOT %IX2.3.56, PT := T#60S);
%ML310.48 := P109C_FS.Q;
(* Rung L277 *)
%ML310.47 := NOT (%QX1.6.0 AND NOT %IX1.3.43 AND %IX2.3.57 AND NOT %ML310.48) OR (%ML310.47 AND NOT %ML1.4 AND NOT %IX1.1.17);
(* Rung L279 *)
%QX2.0.51 := (%QX1.6.0 AND %ML310.47) OR %ML101.0;
(* Rung L281 *)
%QX2.0.52 := ((%QX1.6.0 AND NOT %IX1.3.44) OR %ML101.0) AND NOT %QX2.6.54;
(* Rung L283 *)
IF %QX1.6.0 AND NOT %QX2.0.52 AND ((%QX1.6.2 AND %ML3.50) OR (%QX1.6.3 AND %IX1.3.46)) THEN
    %WW176 := 109;
END_IF;
(* Rung L286 *)
IF %QX1.6.0 AND NOT %QX2.0.52 AND ((%QX1.6.2 AND %ML3.51) OR (%QX1.6.3 AND %IX1.3.45)) THEN
    %WW176 := 0;
END_IF;

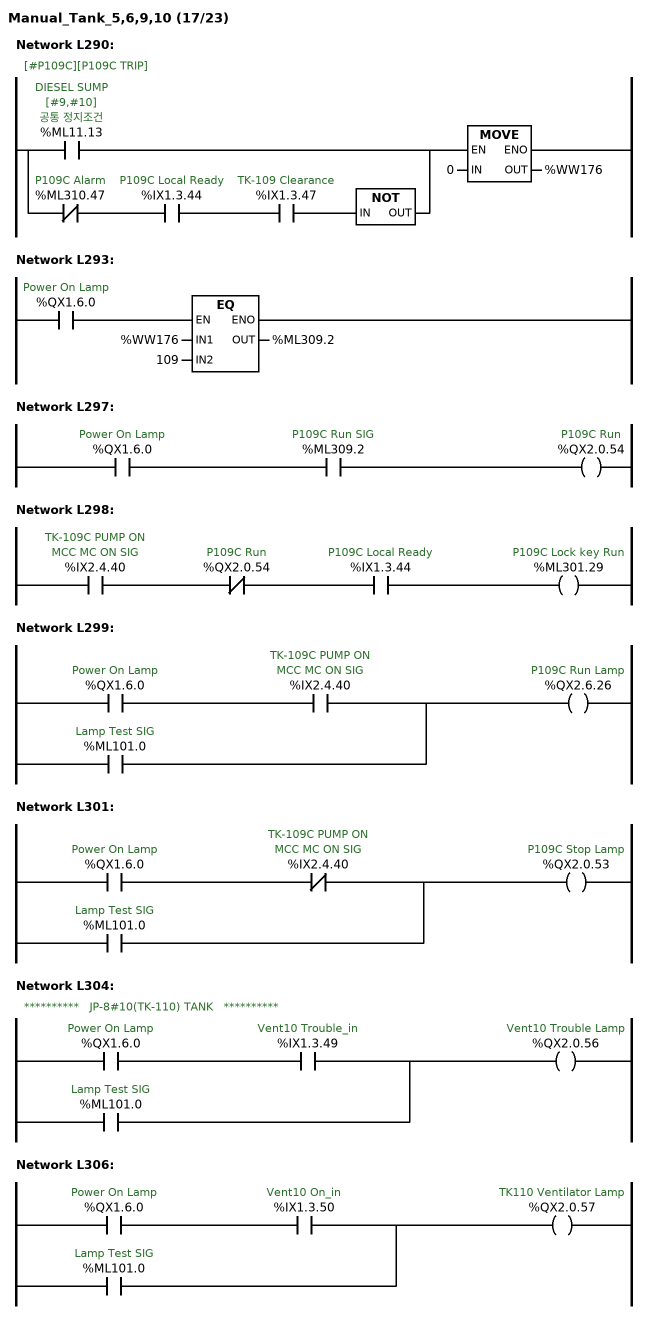
(* [#P109C][P109C TRIP] *)
(* Rung L290 *)
IF %ML11.13 OR (NOT (NOT %ML310.47 AND %IX1.3.44 AND %IX1.3.47)) THEN %WW176 := 0; END_IF;
(* Rung L293 *)
IF %QX1.6.0 THEN %ML309.2 := %WW176 = 109; END_IF;
(* Rung L297 *)
%QX2.0.54 := %QX1.6.0 AND %ML309.2;
(* Rung L298 *)
%ML301.29 := %IX2.4.40 AND NOT %QX2.0.54 AND %IX1.3.44;
(* Rung L299 *)
%QX2.6.26 := (%QX1.6.0 AND %IX2.4.40) OR %ML101.0;
(* Rung L301 *)
%QX2.0.53 := (%QX1.6.0 AND NOT %IX2.4.40) OR %ML101.0;
(* **********   JP-8#10(TK-110) TANK   ********** *)
(* Rung L304 *)
%QX2.0.56 := (%QX1.6.0 AND %IX1.3.49) OR %ML101.0;
(* Rung L306 *)
%QX2.0.57 := (%QX1.6.0 AND %IX1.3.50) OR %ML101.0;

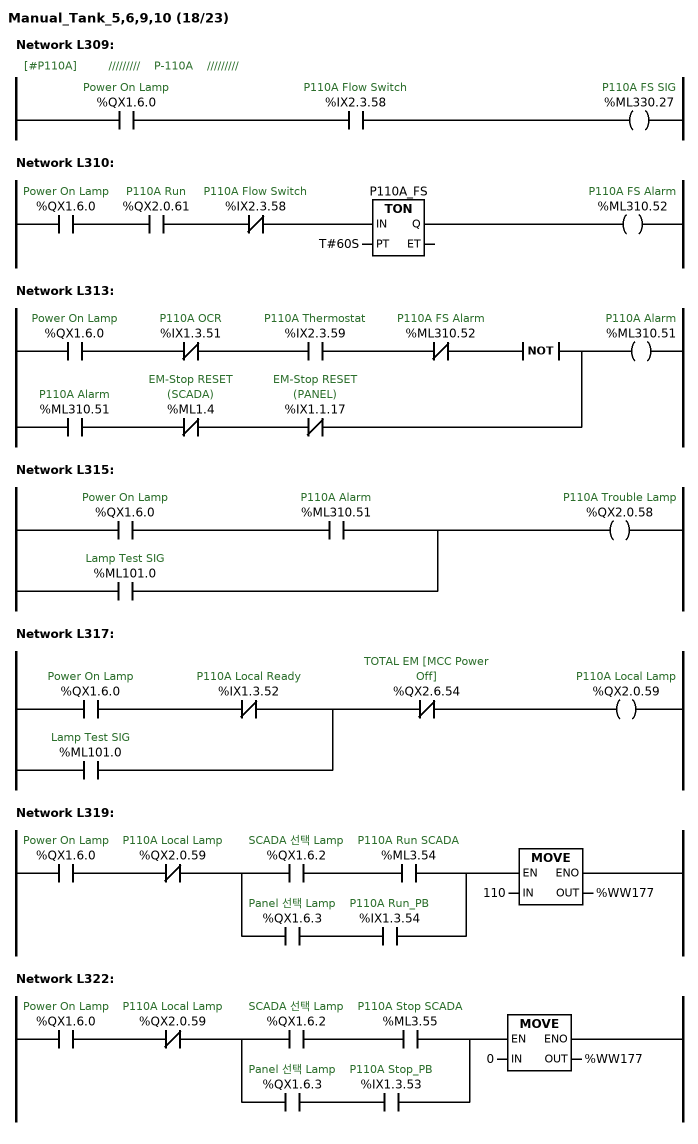
(* [#P110A]         /////////    P-110A    ///////// *)
(* Rung L309 *)
%ML330.27 := %QX1.6.0 AND %IX2.3.58;
(* Rung L310 *)
P110A_FS(IN := %QX1.6.0 AND %QX2.0.61 AND NOT %IX2.3.58, PT := T#60S);
%ML310.52 := P110A_FS.Q;
(* Rung L313 *)
%ML310.51 := NOT (%QX1.6.0 AND NOT %IX1.3.51 AND %IX2.3.59 AND NOT %ML310.52) OR (%ML310.51 AND NOT %ML1.4 AND NOT %IX1.1.17);
(* Rung L315 *)
%QX2.0.58 := (%QX1.6.0 AND %ML310.51) OR %ML101.0;
(* Rung L317 *)
%QX2.0.59 := ((%QX1.6.0 AND NOT %IX1.3.52) OR %ML101.0) AND NOT %QX2.6.54;
(* Rung L319 *)
IF %QX1.6.0 AND NOT %QX2.0.59 AND ((%QX1.6.2 AND %ML3.54) OR (%QX1.6.3 AND %IX1.3.54)) THEN
    %WW177 := 110;
END_IF;
(* Rung L322 *)
IF %QX1.6.0 AND NOT %QX2.0.59 AND ((%QX1.6.2 AND %ML3.55) OR (%QX1.6.3 AND %IX1.3.53)) THEN
    %WW177 := 0;
END_IF;

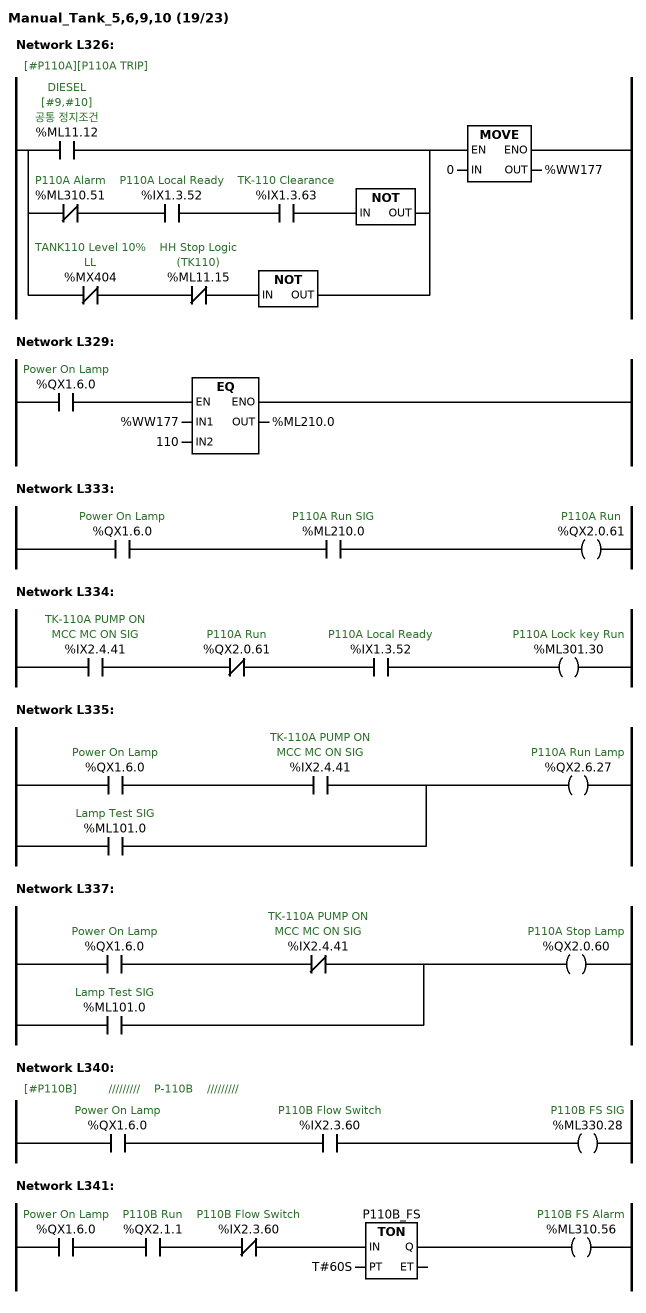
(* [#P110A][P110A TRIP] *)
(* Rung L326 *)
IF %ML11.12 OR (NOT (NOT %ML310.51 AND %IX1.3.52 AND %IX1.3.63)) OR (NOT (NOT %MX404 AND NOT %ML11.15)) THEN
    %WW177 := 0;
END_IF;
(* Rung L329 *)
IF %QX1.6.0 THEN %ML210.0 := %WW177 = 110; END_IF;
(* Rung L333 *)
%QX2.0.61 := %QX1.6.0 AND %ML210.0;
(* Rung L334 *)
%ML301.30 := %IX2.4.41 AND NOT %QX2.0.61 AND %IX1.3.52;
(* Rung L335 *)
%QX2.6.27 := (%QX1.6.0 AND %IX2.4.41) OR %ML101.0;
(* Rung L337 *)
%QX2.0.60 := (%QX1.6.0 AND NOT %IX2.4.41) OR %ML101.0;
(* [#P110B]         /////////    P-110B    ///////// *)
(* Rung L340 *)
%ML330.28 := %QX1.6.0 AND %IX2.3.60;
(* Rung L341 *)
P110B_FS(IN := %QX1.6.0 AND %QX2.1.1 AND NOT %IX2.3.60, PT := T#60S);
%ML310.56 := P110B_FS.Q;

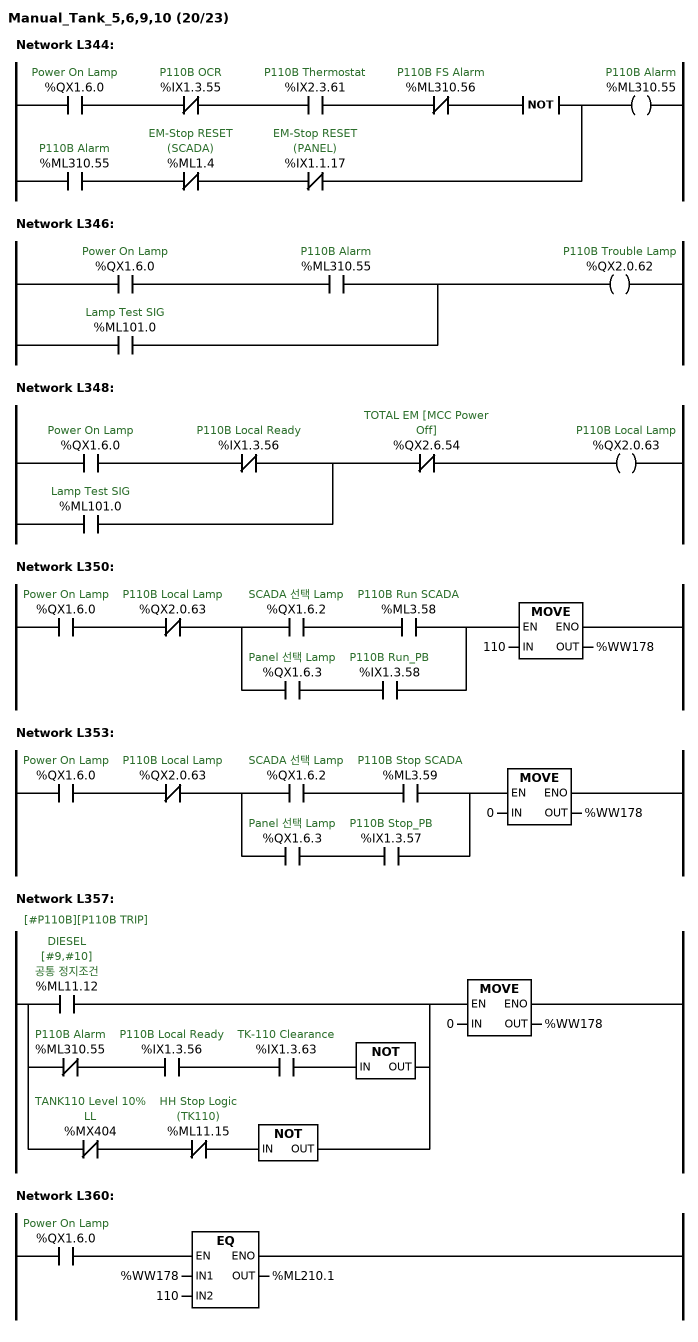
(* Rung L344 *)
%ML310.55 := NOT (%QX1.6.0 AND NOT %IX1.3.55 AND %IX2.3.61 AND NOT %ML310.56) OR (%ML310.55 AND NOT %ML1.4 AND NOT %IX1.1.17);
(* Rung L346 *)
%QX2.0.62 := (%QX1.6.0 AND %ML310.55) OR %ML101.0;
(* Rung L348 *)
%QX2.0.63 := ((%QX1.6.0 AND NOT %IX1.3.56) OR %ML101.0) AND NOT %QX2.6.54;
(* Rung L350 *)
IF %QX1.6.0 AND NOT %QX2.0.63 AND ((%QX1.6.2 AND %ML3.58) OR (%QX1.6.3 AND %IX1.3.58)) THEN
    %WW178 := 110;
END_IF;
(* Rung L353 *)
IF %QX1.6.0 AND NOT %QX2.0.63 AND ((%QX1.6.2 AND %ML3.59) OR (%QX1.6.3 AND %IX1.3.57)) THEN
    %WW178 := 0;
END_IF;
(* [#P110B][P110B TRIP] *)
(* Rung L357 *)
IF %ML11.12 OR (NOT (NOT %ML310.55 AND %IX1.3.56 AND %IX1.3.63)) OR (NOT (NOT %MX404 AND NOT %ML11.15)) THEN
    %WW178 := 0;
END_IF;
(* Rung L360 *)
IF %QX1.6.0 THEN %ML210.1 := %WW178 = 110; END_IF;

